FUNCTION_BLOCK DI_4 (* Function block for a four bit digital input module *)
  (* Standard: 61499-2 *)
  (* Version 0.0, 2014-01-12, 4DIAC-IDE, 4DIAC-Consortium *)
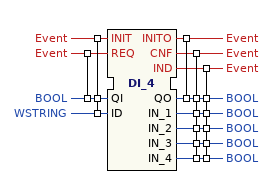
  EVENT_INPUT
    INIT WITH QI, ID; (* Initialization Request *)
    REQ WITH QI; (* Request  update of the input values *)
  END_EVENT
  EVENT_OUTPUT
    INITO WITH QO; (* Initialization Confirm *)
    CNF WITH QO, IN_1, IN_2, IN_3, IN_4; (* Input values updated *)
    IND WITH QO, IN_1, IN_2, IN_3, IN_4; (* Indication on input value changes *)
  END_EVENT
  VAR_INPUT
    QI : BOOL; (* Input event qualifier *)
    ID : WSTRING; (* Identifier for the input module *)
  END_VAR
  VAR_OUTPUT
    QO : BOOL; (* Output event qualifier *)
    IN_1 : BOOL;
    IN_2 : BOOL;
    IN_3 : BOOL;
    IN_4 : BOOL;
  END_VAR
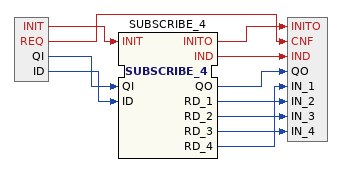
  FBS
    SUBSCRIBE_4 : SUBSCRIBE_4;
  END_FBS
  EVENT_CONNECTIONS
    REQ TO CNF;
    INIT TO SUBSCRIBE_4.INIT;
    SUBSCRIBE_4.INITO TO INITO;
    SUBSCRIBE_4.IND TO IND;
  END_CONNECTIONS
  DATA_CONNECTIONS
    QI TO SUBSCRIBE_4.QI;
    ID TO SUBSCRIBE_4.ID;
    SUBSCRIBE_4.QO TO QO;
    SUBSCRIBE_4.RD_1 TO IN_1;
    SUBSCRIBE_4.RD_2 TO IN_2;
    SUBSCRIBE_4.RD_3 TO IN_3;
    SUBSCRIBE_4.RD_4 TO IN_4;
  END_CONNECTIONS
END_FUNCTION_BLOCK
